{attribute 'GeneratedUsingTerminal: EL2262--0000'}
{attribute addProperty BoxType "EL2262--0000"}
{attribute addProperty Id "OutputAT %Q*BYTE1"}
{attribute addProperty CRC "1011221447"}
{attribute addProperty Size "1"}
TYPE Sample_3C4603C7 :
STRUCT
	{attribute addProperty Name "Output"}
	Output AT %Q* : BYTE;
END_STRUCT
END_TYPE

(* stored: Version 1.2.0.0, ProductVersion 3.1.4024.9
   DUT Sample_3C4603C7: Id {80808390-8d49-410e-9cab-191849508935} *)
